TYPE Homing :
STRUCT
	Mode			:		HomingMode;
	FlagType		:		HomeFlagType;
	bHomeInput		:		BOOL;
	rOffset			:		REAL;
	rVelocity		:		REAL;
	rTorque			:		REAL;
END_STRUCT
END_TYPE

(* stored: Version 1.1.0.1, ProductVersion 3.1.4024.6
   DUT Homing: Id {a875da55-0f01-4e05-a482-9f572e0b6239} *)
